FUNCTION BuildStringInline : REFERENCE TO StringBuilder
VAR_INPUT
	value : T_MaxString;
END_VAR
VAR_STAT
	builder : StringBuilder;
END_VAR

builder.Clear();

builder.Append(value);

BuildStringInline := builder;

END_FUNCTION

(* stored: Version 1.1.0.1, ProductVersion 3.1.4024.12
   POU BuildStringInline: Id {4bb7c327-72de-4bac-bd0a-0c4baff7eb29}, SpecialFunc None *)
